Yaskawa INFORM job: X4-SCHODKI_ZEW.JBI

/JOB
//NAME X4-SCHODKI_ZEW
//POS
///NPOS 224,224,224,10,0,0
///TOOL 0
///POSTYPE PULSE
///PULSE
C00000=21160,-126487,-99095,6220,53097,19917
C00001=122314,-84956,-84267,5758,65294,20346
C00002=113867,-2788,-32259,11364,77586,-20622
C00003=111699,9606,-11794,12514,71800,-21939
C00004=110873,16102,-4909,12893,71047,-22311
C00005=111426,18220,-2948,12689,70847,-22135
C00006=111334,17863,-3281,12723,70881,-22164
C00007=111334,17842,-1921,12786,70054,-22254
C00008=111688,13758,-7042,12574,71029,-22022
C00009=137921,23655,2193,-26065,80546,13065
C00010=138187,30095,8478,-26164,80127,13260
C00011=137141,31636,10013,-25924,79665,12972
C00012=137283,31426,9804,-25956,79727,13011
C00013=137283,31447,11085,-26011,79025,13166
C00014=137811,24810,3269,-26040,80453,13045
C00015=130093,15204,-5597,-17076,73087,3422
C00016=130254,16762,-4164,-17139,73044,3486
C00017=130499,11823,-8660,-17205,73314,3535
C00018=136657,16032,-4835,-19303,74485,5576
C00019=136779,34044,12201,-19450,73350,5806
C00020=136367,37287,16065,-19383,72578,5782
C00021=135529,38270,17077,-19116,72272,5524
C00022=135735,38345,17156,-19186,72312,5593
C00023=135735,38391,18179,-19247,71738,5687
C00024=136093,38073,17157,-19317,72259,5733
C00025=136821,38987,18103,-19565,72324,5991
C00026=137234,41236,20445,-19732,72152,6174
C00027=137468,37941,16529,-19737,72884,6137
C00028=139273,33119,8814,-10616,74138,14432
C00029=138400,39162,15428,-10360,73077,14220
C00030=137624,40756,17090,-10099,72782,13973
C00031=137810,40443,16764,-10163,72844,14033
C00032=137810,40460,18419,-10216,71849,14119
C00033=138377,33107,10032,-10341,73283,14197
C00034=129933,32626,9546,1459,71562,3103
C00035=130107,34413,11352,1398,71367,3162
C00036=130344,28976,5916,1305,71915,3250
C00037=134876,30968,7890,-396,71698,4822
C00038=142592,70732,50995,-12851,68399,16892
C00039=141830,71409,51797,-12602,68137,16639
C00040=142006,70894,51186,-12652,68274,16689
C00041=142006,71149,52557,-12712,67578,16765
C00042=142006,71007,51815,-12679,67954,16725
C00043=142747,76515,58410,-13043,66871,17119
C00044=142702,66110,44987,-12780,69711,16790
C00045=130401,22900,-3912,9781,74013,14096
C00046=130750,-77898,-76934,10038,67211,13654
C00047=128341,-94500,-64478,15665,37561,8814
C00048=125354,-34494,-33676,16070,41961,8103
C00049=123908,-22688,-35224,-7311,60763,8117
C00050=115329,1774,-22996,-8583,68206,33205
C00051=113811,6923,-16554,-7934,66753,32769
C00052=112938,8598,-15088,-7517,66630,32466
C00053=113357,7607,-15958,-7718,66694,32611
C00054=113357,7474,-14642,-7767,65823,32669
C00055=113357,7562,-15559,-7732,66427,32629
C00056=114674,8046,-17033,-9196,71995,10105
C00057=114277,9137,-16073,-9034,71921,9973
C00058=114994,10710,-14679,-9331,71949,10219
C00059=115929,5782,-19714,-10610,72890,11247
C00060=114914,9168,-18033,-20160,83408,25507
C00061=114509,10465,-16323,-20060,82947,25443
C00062=114509,10278,-15209,-20089,82211,25564
C00063=114509,10430,-16126,-20066,82816,25464
C00064=113574,12027,-14696,-19812,82540,25184
C00065=113966,9476,-16971,-19916,82715,25292
C00066=109195,41890,2270,-19889,88323,22522
C00067=109420,41611,2136,-14547,83651,24420
C00068=109633,43097,3705,-14621,83493,24508
C00069=110073,47498,8361,-9922,80898,20177
C00070=110340,48514,8983,-10012,81065,20250
C00071=109875,50139,10594,-6927,80049,17487
C00072=111642,41129,-2073,-7513,83338,17864
C00073=120740,-4591,-30289,-15267,55452,23675
C00074=120758,-111403,-89341,-20679,37744,27189
C00075=120758,-111403,-89341,-20679,37744,27189
C00076=97140,-41370,-74515,11864,90116,-15742
C00077=93918,-16818,-51601,15265,90472,-19448
C00078=96838,-21310,-54909,14446,89719,-18600
C00079=97144,-22320,-55662,14359,89616,-18514
C00080=98771,-24881,-57497,13895,89173,-18041
C00081=115828,-29996,-61044,-7286,86100,2495
C00082=121364,-24267,-57094,-13933,89260,9154
C00083=125066,-13537,-49221,-14991,90516,10198
C00084=125405,-12324,-48437,-15087,90711,10281
C00085=127775,-3453,-41245,-15747,91251,10973
C00086=117906,-11103,-47413,-1372,86513,-3179
C00087=107817,-4833,-42392,13913,90158,-17947
C00088=111065,-8601,-45456,12965,89620,-16971
C00089=111228,-9142,-45834,12917,89553,-16926
C00090=113235,-11504,-47787,12324,89257,-16321
C00091=116129,-16038,-53218,11461,89860,-15351
C00092=132129,3503,-37461,731,88042,-5165
C00093=134839,10104,-29765,-1476,86561,-3078
C00094=133535,10494,-29542,-1044,86604,-3481
C00095=133472,10527,-29512,-1023,86602,-3500
C00096=132997,13157,-27039,-5636,86965,851
C00097=131112,-12606,-50888,-7793,88905,29033
C00098=129834,-10958,-47906,-7386,87816,28703
C00099=133351,1378,-37957,-8503,88347,29764
C00100=133639,2898,-36665,-8594,88358,29852
C00101=132895,14544,-26435,-2898,86896,24452
C00102=133144,15405,-25686,-2979,86883,24528
C00103=133588,9909,-35564,-3125,90148,24585
C00104=114600,-38617,-66572,24501,76796,21744
C00105=88804,-102668,-113384,34072,81784,13502
C00106=-3643,-76224,-106676,-19950,71810,-76872
C00107=-6047,-95755,-92046,14751,98253,-9605
C00108=-2299,-70459,-84112,3705,91093,-18065
C00109=-2299,-70459,-84112,3705,91093,-18065
C00110=-2299,-70459,-84112,3705,91093,-18065
C00111=-2299,-70459,-84112,3705,91093,-18065
C00112=61951,-108908,-90353,7974,21769,-53190
C00113=44975,-75191,-76287,54105,62461,-71292
C00114=78581,-58710,-61930,31634,35162,-55381
C00115=95060,-56001,-58325,12610,29924,-73279
C00116=99699,-51031,-54888,6140,29822,-70179
C00117=99897,-48307,-53304,5791,30229,-70010
C00118=100054,-49149,-53798,5600,30089,-69920
C00119=100054,-49034,-52503,5728,29355,-69986
C00120=100054,-49149,-53798,5600,30089,-69920
C00121=86412,-51164,-57714,27133,38899,-75152
C00122=76272,-10487,-35891,41089,67840,-66679
C00123=77011,-10638,-36009,40769,67508,-66483
C00124=76817,-10362,-35793,40851,67601,-66531
C00125=76817,-10560,-34912,41019,67109,-66737
C00126=76817,-10362,-35793,40851,67601,-66531
C00127=75718,7442,-20978,41322,68120,-66813
C00128=76464,7847,-20622,41001,67775,-66619
C00129=76126,7559,-20874,41146,67933,-66706
C00130=76126,7348,-19931,41325,67409,-66927
C00131=76126,7559,-20874,41146,67933,-66706
C00132=91627,-14375,-38555,867,50575,-46141
C00133=91624,-12364,-37017,870,50664,-46141
C00134=91625,-13152,-37622,869,50631,-46141
C00135=91625,-13360,-36631,878,49914,-46147
C00136=91625,-13152,-37622,869,50631,-46141
C00137=68864,9101,-19550,42290,68970,-68812
C00138=70480,17607,-11844,41698,67948,-68513
C00139=71103,18297,-11202,41441,67635,-68362
C00140=70696,17763,-11700,41608,67844,-68460
C00141=70696,17560,-10741,41791,67318,-68687
C00142=70696,17763,-11700,41608,67844,-68460
C00143=71865,37445,7605,38393,62836,-66759
C00144=72519,37882,8057,38094,62514,-66586
C00145=71865,37445,7605,38393,62836,-66759
C00146=71865,37288,8698,38629,62241,-66997
C00147=71865,37445,7605,38393,62836,-66759
C00148=69589,28187,-3550,38858,65482,-66746
C00149=81736,18570,-13478,9629,55098,-51480
C00150=92480,21393,-8443,-18166,53536,-36270
C00151=92406,23699,-6245,-18150,53360,-36270
C00152=92480,21393,-8443,-18166,53536,-36270
C00153=92480,21153,-7249,-18365,52720,-36120
C00154=92480,21393,-8443,-18166,53536,-36270
C00155=66161,2763,-24906,35901,59847,-65565
C00156=8779,-64345,-72223,57070,85976,-80913
C00157=8779,-64345,-72223,57070,85976,-80913
C00158=80709,2938,-29836,37807,72072,-57205
C00159=104099,16313,-17981,36138,70132,-56262
C00160=141757,27909,-6366,14089,61839,-44283
C00161=141757,27617,-5405,14183,61121,-44376
C00162=141757,27909,-6366,14089,61839,-44283
C00163=142084,29535,-4762,13913,61639,-44186
C00164=141757,27909,-6366,14089,61839,-44283
C00165=134298,42766,7339,18583,62496,-46981
C00166=136587,44887,8503,12300,63619,-46934
C00167=136587,44658,9247,12359,63057,-46997
C00168=136587,44887,8503,12300,63619,-46934
C00169=137255,47131,10909,11951,63202,-46735
C00170=136587,44887,8503,12300,63619,-46934
C00171=137657,47095,11743,9838,62197,-45465
C00172=138989,44169,8634,9022,62453,-44958
C00173=139465,42914,7769,8751,62290,-44797
C00174=139736,38942,3601,15550,64524,-48931
C00175=140033,37764,2383,15370,64612,-48812
C00176=142152,32374,-3332,17000,65924,-49772
C00177=136320,25956,-14717,19617,70677,-51083
C00178=115846,-52963,-75028,29682,73275,-57924
C00179=37442,-83575,-86281,52659,88245,-87706
C00180=33903,-112886,-95665,42735,53090,-80159
C00181=69561,-59751,-72923,16095,52051,-63361
C00182=88044,4124,-27726,-14416,55568,-38396
C00183=89480,30550,-2469,-15773,59241,-38542
C00184=89566,29946,-3118,-13987,58895,-39575
C00185=89868,30274,-2806,-13508,58764,-39848
C00186=89813,28581,-4483,-7975,57782,-42956
C00187=83888,29903,-3137,7775,57604,-51754
C00188=72316,13965,-19527,34407,71386,-67147
C00189=73909,13977,-18764,33784,70394,-66825
C00190=73971,16364,-16409,33799,70187,-66867
C00191=73672,28324,-4910,34113,69520,-67204
C00192=73857,29288,-3960,34049,69373,-67175
C00193=73190,47231,14588,34804,67803,-67970
C00194=76539,39499,6435,26306,62774,-62506
C00195=71407,-68,-33227,28174,68008,-63188
C00196=92287,-5015,-35072,-6189,59116,-43997
C00197=93582,-5318,-35114,-7054,59088,-43517
C00198=94768,-5424,-35240,-7833,59212,-43086
C00199=95122,-4999,-34965,-8061,59297,-42962
C00200=98977,-4910,-34893,-10570,59720,-41566
C00201=89817,-2997,-33375,10480,59755,-53225
C00202=87165,-16267,-43774,12233,59696,-54222
C00203=74457,-13339,-39679,39309,71456,-68037
C00204=78370,-12635,-39382,37625,69939,-66937
C00205=80519,-10300,-39984,32672,71010,-66549
C00206=79797,2903,-29087,32982,71339,-66737
C00207=79943,3599,-28462,32921,71264,-66703
C00208=82505,7061,-25304,26471,66621,-62758
C00209=86409,1492,-30136,17739,62740,-57641
C00210=82783,-10794,-40788,19813,63755,-58809
C00211=89567,-44228,-57976,15859,46252,-64914
C00212=95371,-48907,-52544,12165,29960,-73065
C00213=96871,-48956,-52574,10129,29748,-72091
C00214=98013,-48924,-52556,8555,29621,-71337
C00215=98537,-48530,-52441,7796,29699,-70974
C00216=102207,-48035,-52053,2674,29480,-68529
C00217=94327,-44885,-50172,28699,34004,-81028
C00218=94609,-45389,-50476,28446,33845,-80908
C00219=90036,-53113,-58492,32420,36321,-82805
C00220=51114,-81290,-74278,61960,52593,-60278
C00221=6076,-109546,-85200,71251,79672,-70600
C00222=6076,-109546,-85200,71251,79672,-70600
C00223=6076,-109546,-85200,-4239,76823,-70600
BC00000=277643,516186,172088
BC00001=328181,496789,172088
BC00002=328180,496788,172085
BC00003=328180,496788,172085
BC00004=328180,496788,172085
BC00005=328180,496788,172085
BC00006=328180,496788,172085
BC00007=328180,496788,172085
BC00008=328180,496788,172085
BC00009=328180,496788,172085
BC00010=328180,496788,172085
BC00011=328180,496788,172085
BC00012=328180,496788,172085
BC00013=328180,496788,172085
BC00014=328180,496788,172085
BC00015=328180,496788,172085
BC00016=328180,496788,172085
BC00017=328180,496788,172085
BC00018=328180,496788,172085
BC00019=328180,496788,172085
BC00020=328180,496788,172085
BC00021=328180,496788,172085
BC00022=328180,496788,172085
BC00023=328180,496788,172085
BC00024=328180,496788,172085
BC00025=328180,496788,172085
BC00026=328180,496788,172085
BC00027=328180,496788,172085
BC00028=328180,496788,172085
BC00029=328180,496788,172085
BC00030=328180,496788,172085
BC00031=328180,496788,172085
BC00032=328180,496788,172085
BC00033=328180,496788,172085
BC00034=328180,496788,172085
BC00035=328180,496788,172085
BC00036=328180,496788,172085
BC00037=328180,496788,172085
BC00038=328180,496788,172085
BC00039=328180,496788,172085
BC00040=328180,496788,172085
BC00041=328180,496788,172085
BC00042=328180,496788,172085
BC00043=328180,496788,172085
BC00044=328180,496788,172085
BC00045=328180,496788,172085
BC00046=328180,496788,172085
BC00047=194416,502028,172085
BC00048=194416,502028,172085
BC00049=173311,425006,172085
BC00050=173311,425006,140819
BC00051=173311,425006,140819
BC00052=173311,425006,140819
BC00053=173311,425006,140819
BC00054=173311,425006,140819
BC00055=173311,425006,140819
BC00056=173311,425006,140819
BC00057=173311,425006,140819
BC00058=173311,425006,140819
BC00059=173311,425006,140819
BC00060=173311,425006,140819
BC00061=173311,425006,140819
BC00062=173311,425006,140819
BC00063=173311,425006,140819
BC00064=173311,425006,140819
BC00065=173311,425006,140819
BC00066=158492,452266,59327
BC00067=158492,452266,59327
BC00068=158492,452266,59327
BC00069=158492,452266,59327
BC00070=158492,452266,59327
BC00071=158492,452266,59327
BC00072=158492,452266,59327
BC00073=158492,452266,59327
BC00074=158492,507957,59327
BC00075=293306,507957,59327
BC00076=293305,437676,59324
BC00077=293305,437676,59324
BC00078=293305,437676,59324
BC00079=293305,437676,59324
BC00080=293305,437676,59324
BC00081=293305,437676,59324
BC00082=293305,437676,59324
BC00083=293305,437676,59324
BC00084=293305,437676,59324
BC00085=293305,437676,59324
BC00086=293305,437676,59324
BC00087=293305,437676,59324
BC00088=293305,437676,59324
BC00089=293305,437676,59324
BC00090=293305,437676,59324
BC00091=293305,437676,59324
BC00092=293305,437676,59324
BC00093=293305,437676,59324
BC00094=293305,437676,59324
BC00095=293305,437676,59324
BC00096=293305,437676,59324
BC00097=293305,437676,59324
BC00098=293305,437676,59324
BC00099=293305,437676,59324
BC00100=293305,437676,59324
BC00101=293305,437676,59324
BC00102=293305,437676,59324
BC00103=293305,437676,59324
BC00104=293305,437676,59324
BC00105=293305,491548,59324
BC00106=199448,515539,1075137
BC00107=95028,515070,919110
BC00108=123826,515279,972180
BC00109=123826,515279,972180
BC00110=123826,515279,972180
BC00111=44761,462630,27794
BC00112=44761,462630,27794
BC00113=44761,462630,27793
BC00114=44761,462630,27793
BC00115=44761,462630,27793
BC00116=44761,462630,27793
BC00117=44761,462630,27793
BC00118=44761,462630,27793
BC00119=44761,462630,27793
BC00120=44761,462630,27793
BC00121=44761,462630,27793
BC00122=44761,462630,27793
BC00123=44761,462630,27793
BC00124=44761,462630,27793
BC00125=44761,462630,27793
BC00126=44761,462630,27793
BC00127=44761,462630,27793
BC00128=44761,462630,27793
BC00129=44761,462630,27793
BC00130=44761,462630,27793
BC00131=44761,462630,27793
BC00132=44761,462630,27793
BC00133=44761,462630,27793
BC00134=44761,462630,27793
BC00135=44761,462630,27793
BC00136=44761,462630,27793
BC00137=44761,462630,27793
BC00138=44761,462630,27793
BC00139=44761,462630,27793
BC00140=44761,462630,27793
BC00141=44761,462630,27793
BC00142=44761,462630,27793
BC00143=44761,462630,27793
BC00144=44761,462630,27793
BC00145=44761,462630,27793
BC00146=44761,462630,27793
BC00147=44761,462630,27793
BC00148=44761,462630,27793
BC00149=44761,462630,27793
BC00150=44761,462630,27793
BC00151=44761,462630,27793
BC00152=44761,462630,27793
BC00153=44761,462630,27793
BC00154=44761,462630,27793
BC00155=44761,462630,27792
BC00156=44761,462630,27792
BC00157=202931,462630,27792
BC00158=202931,462630,27792
BC00159=222940,462630,27792
BC00160=308656,462630,27792
BC00161=308656,462630,27792
BC00162=308656,462630,27792
BC00163=308656,462630,27792
BC00164=308656,462630,27792
BC00165=308656,462630,27792
BC00166=308656,462630,27792
BC00167=308656,462630,27792
BC00168=308656,462630,27792
BC00169=308656,462630,27792
BC00170=308656,462630,27792
BC00171=308656,462630,27792
BC00172=308656,462630,27792
BC00173=308656,462630,27792
BC00174=308656,462630,27792
BC00175=308656,462630,27792
BC00176=308656,462630,27792
BC00177=308656,462630,27792
BC00178=308656,462630,27791
BC00179=194109,459376,27791
BC00180=59950,457329,27792
BC00181=59950,457329,27792
BC00182=44761,462630,27793
BC00183=44761,462629,27792
BC00184=44761,462629,27792
BC00185=44761,462629,27792
BC00186=44761,462629,27792
BC00187=44761,462629,27792
BC00188=44761,462629,27792
BC00189=44761,462629,27792
BC00190=44761,462629,27792
BC00191=44761,462629,27792
BC00192=44761,462629,27792
BC00193=44761,462629,27792
BC00194=44761,462629,27792
BC00195=44761,462629,27792
BC00196=44761,462629,27792
BC00197=44761,462629,27792
BC00198=44761,462629,27792
BC00199=44761,462629,27792
BC00200=44761,462629,27792
BC00201=44761,462629,27792
BC00202=44761,462629,27792
BC00203=44761,462629,27792
BC00204=44761,462629,27792
BC00205=44761,462629,27792
BC00206=44761,462629,27792
BC00207=44761,462629,27792
BC00208=44761,462629,27792
BC00209=44761,462629,27792
BC00210=44761,462629,27792
BC00211=44761,462629,27792
BC00212=44761,462630,27793
BC00213=44761,462630,27793
BC00214=44761,462630,27793
BC00215=44761,462630,27793
BC00216=44761,462630,27793
BC00217=44761,462630,27793
BC00218=44761,462630,27793
BC00219=44761,462630,27793
BC00220=44761,462630,27793
BC00221=44761,546100,27793
BC00222=44761,546100,27793
BC00223=44761,546100,971290
EC00000=798156,-183832
EC00001=798156,-183832
EC00002=798153,-183831
EC00003=798153,-183831
EC00004=798153,-183831
EC00005=798153,-183831
EC00006=798153,-183831
EC00007=798153,-183831
EC00008=798153,-183831
EC00009=798153,-183831
EC00010=798153,-183831
EC00011=798153,-183831
EC00012=798153,-183831
EC00013=798153,-183831
EC00014=798153,-183831
EC00015=798153,-183831
EC00016=798153,-183831
EC00017=798153,-183831
EC00018=798153,-183831
EC00019=798153,-183831
EC00020=798153,-183831
EC00021=798153,-183831
EC00022=798153,-183831
EC00023=798153,-183831
EC00024=798153,-183831
EC00025=798153,-183831
EC00026=798153,-183831
EC00027=798153,-183831
EC00028=798153,-183831
EC00029=798153,-183831
EC00030=798153,-183831
EC00031=798153,-183831
EC00032=798153,-183831
EC00033=798153,-183831
EC00034=798153,-183831
EC00035=798153,-183831
EC00036=798153,-183831
EC00037=798153,-183831
EC00038=798153,-183831
EC00039=798153,-183831
EC00040=798153,-183831
EC00041=798153,-183831
EC00042=798153,-183831
EC00043=798153,-183831
EC00044=798153,-183831
EC00045=798153,-183831
EC00046=798153,-183831
EC00047=798153,-183831
EC00048=798153,-183831
EC00049=798153,-183831
EC00050=798153,-183831
EC00051=798153,-183831
EC00052=798153,-183831
EC00053=798153,-183831
EC00054=798153,-183831
EC00055=798153,-183831
EC00056=798153,-183831
EC00057=798153,-183831
EC00058=798153,-183831
EC00059=798153,-183831
EC00060=798153,-183831
EC00061=798153,-183831
EC00062=798153,-183831
EC00063=798153,-183831
EC00064=798153,-183831
EC00065=798153,-183831
EC00066=798153,-183831
EC00067=798153,-183831
EC00068=798153,-183831
EC00069=798153,-183831
EC00070=798153,-183831
EC00071=798153,-183831
EC00072=798153,-183831
EC00073=798153,-183831
EC00074=798153,-183831
EC00075=798153,-183831
EC00076=798151,-183830
EC00077=798151,-183830
EC00078=798151,-183830
EC00079=798151,-183830
EC00080=798151,-183830
EC00081=798151,-183830
EC00082=798151,-183830
EC00083=798151,-183830
EC00084=798151,-183830
EC00085=798151,-183830
EC00086=798151,-183830
EC00087=798151,-183830
EC00088=798151,-183830
EC00089=798151,-183830
EC00090=798151,-183830
EC00091=798151,-183830
EC00092=798151,-183830
EC00093=798151,-183830
EC00094=798151,-183830
EC00095=798151,-183830
EC00096=798151,-183830
EC00097=798151,-183830
EC00098=798151,-183830
EC00099=798151,-183830
EC00100=798151,-183830
EC00101=798151,-183830
EC00102=798151,-183830
EC00103=798151,-183830
EC00104=798151,-183830
EC00105=798151,-183830
EC00106=798151,-183830
EC00107=798156,-183832
EC00108=322978,-183832
EC00109=357094,925242
EC00110=800604,925242
EC00111=800604,925242
EC00112=800604,925242
EC00113=800603,925242
EC00114=800603,925242
EC00115=800603,925242
EC00116=800603,925242
EC00117=800603,925242
EC00118=800603,925242
EC00119=800603,925242
EC00120=800603,925242
EC00121=800603,925242
EC00122=800603,925242
EC00123=800603,925242
EC00124=800603,925242
EC00125=800603,925242
EC00126=800603,925242
EC00127=800603,925242
EC00128=800603,925242
EC00129=800603,925242
EC00130=800603,925242
EC00131=800603,925242
EC00132=800603,925242
EC00133=800603,925242
EC00134=800603,925242
EC00135=800603,925242
EC00136=800603,925242
EC00137=800603,925242
EC00138=800603,925242
EC00139=800603,925242
EC00140=800603,925242
EC00141=800603,925242
EC00142=800603,925242
EC00143=800603,925242
EC00144=800603,925242
EC00145=800603,925242
EC00146=800603,925242
EC00147=800603,925242
EC00148=800603,925242
EC00149=800601,925240
EC00150=800600,925239
EC00151=800600,925239
EC00152=800600,925239
EC00153=800600,925239
EC00154=800600,925239
EC00155=800598,925238
EC00156=800598,925238
EC00157=800598,925238
EC00158=800598,925238
EC00159=800598,925238
EC00160=800598,925238
EC00161=800598,925238
EC00162=800598,925238
EC00163=800598,925238
EC00164=800598,925238
EC00165=800598,925238
EC00166=800598,925238
EC00167=800598,925238
EC00168=800598,925238
EC00169=800598,925238
EC00170=800598,925238
EC00171=800598,925238
EC00172=800598,925238
EC00173=800598,925238
EC00174=800598,925238
EC00175=800598,925238
EC00176=800598,925238
EC00177=800598,925238
EC00178=800591,925233
EC00179=800591,925233
EC00180=800596,925236
EC00181=800596,925236
EC00182=800600,925239
EC00183=800597,925236
EC00184=800597,925236
EC00185=800597,925236
EC00186=800597,925236
EC00187=800597,925236
EC00188=800597,925236
EC00189=800597,925236
EC00190=800597,925236
EC00191=800597,925236
EC00192=800597,925236
EC00193=800597,925236
EC00194=800597,925236
EC00195=800597,925236
EC00196=800597,925236
EC00197=800597,925236
EC00198=800597,925236
EC00199=800597,925236
EC00200=800597,925236
EC00201=800597,925236
EC00202=800597,925236
EC00203=800597,925236
EC00204=800597,925236
EC00205=800597,925236
EC00206=800597,925236
EC00207=800597,925236
EC00208=800597,925236
EC00209=800597,925236
EC00210=800594,925234
EC00211=800598,925238
EC00212=800603,925242
EC00213=800603,925242
EC00214=800603,925242
EC00215=800603,925242
EC00216=800603,925242
EC00217=800603,925242
EC00218=800603,925242
EC00219=800603,925242
EC00220=800603,925242
EC00221=800603,925242
EC00222=-11362,925242
EC00223=-11362,925242
///POSTYPE BASE
///RECTAN
///RCONF 0,0,0,0,1,0,0,0,0,0,0,0,0,0,0,0,0,0,0,0,0,0,0,0
P00006=2.006,1.622,-0.565,0.0000,0.0000,0.0000
P00021=0.073,2.058,-0.109,0.0000,0.0000,0.0000
P00022=2.006,1.622,-0.565,0.0000,0.0000,0.0000
///RCONF 0,0,0,0,0,0,0,0,0,0,0,0,0,0,0,0,0,0,0,0,0,0,0,0
P00023=-2.957,-4.083,2.762,0.0000,0.0000,0.0000
P00024=-1.466,-0.226,-0.419,0.0000,0.0000,0.0000
P00025=3.643,0.007,-2.585,0.0000,0.0000,0.0000
P00026=2.644,0.055,-2.583,0.0000,0.0000,0.0000
P00027=2.278,0.099,-4.210,0.0000,0.0000,0.0000
P00028=-1.778,-0.182,-2.050,0.0000,0.0000,0.0000
P00029=1.749,4.006,-0.261,0.0000,0.0000,0.0000
//INST
///DATE 2024/11/26 12:08
///ATTR SC,RW
///GROUP1 RB1,BS1
///GROUP2 ST1
NOP
MOVJ C00000 BC00000 VJ=100.00  +MOVJ EC00000 VJ=100.00
MOVJ C00001 BC00001 VJ=100.00  +MOVJ EC00001 VJ=100.00
MOVJ C00002 BC00002 VJ=100.00  +MOVJ EC00002 VJ=100.00
SMOVL C00003 BC00003 V=833.3  +MOVJ EC00003
SMOVL C00004 BC00004 V=166.7  +MOVJ EC00004
SREFP 3 C00005 BC00005  +REFP EC00005
CALL JOB:SEARCH-R1-S13D
SET P021 P006
SFTON3D P021
SMOVL C00006 BC00006 V=166.7  +MOVJ EC00006
SREFP 3 C00007 BC00007  +REFP EC00007
CALL JOB:SEARCH-R1-S13D
SET P021 P006
SFTON3D P021
SMOVL C00008 BC00008 V=166.7  +MOVJ EC00008
SFTOF3D
SMOVL C00009 BC00009 V=833.3  +MOVJ EC00009
SMOVL C00010 BC00010 V=166.7  +MOVJ EC00010
SREFP 3 C00011 BC00011  +REFP EC00011
CALL JOB:SEARCH-R1-S13D
SET P022 P006
SFTON3D P022
SMOVL C00012 BC00012 V=166.7  +MOVJ EC00012
SREFP 3 C00013 BC00013  +REFP EC00013
CALL JOB:SEARCH-R1-S13D
SET P022 P006
SFTON3D P022
SMOVL C00014 BC00014 V=166.7  +MOVJ EC00014
SMOVL C00015 BC00015 V=166.7  +MOVJ EC00015
SREFP 3 C00016 BC00016  +REFP EC00016
CALL JOB:SEARCH-R1-S13D
SET P022 P006
SFTON3D P022
SMOVL C00017 BC00017 V=166.7  +MOVJ EC00017
SFTOF3D
SMOVL C00018 BC00018 V=500.0  +MOVJ EC00018
SMOVL C00019 BC00019 V=500.0  +MOVJ EC00019
SMOVL C00020 BC00020 V=166.7  +MOVJ EC00020
SREFP 3 C00021 BC00021  +REFP EC00021
CALL JOB:SEARCH-R1-S13D
SET P023 P006
SFTON3D P023
SMOVL C00022 BC00022 V=166.7  +MOVJ EC00022
SREFP 3 C00023 BC00023  +REFP EC00023
CALL JOB:SEARCH-R1-S13D
SET P023 P006
SFTON3D P023
SMOVL C00024 BC00024 V=166.7  +MOVJ EC00024
SMOVL C00025 BC00025 V=166.7  +MOVJ EC00025
SREFP 3 C00026 BC00026  +REFP EC00026
CALL JOB:SEARCH-R1-S13D
SET P023 P006
SFTON3D P023
SMOVL C00027 BC00027 V=166.7  +MOVJ EC00027
SFTOF3D
SMOVL C00028 BC00028 V=333.3  +MOVJ EC00028
SMOVL C00029 BC00029 V=166.7  +MOVJ EC00029
SREFP 3 C00030 BC00030  +REFP EC00030
CALL JOB:SEARCH-R1-S13D
SET P024 P006
SFTON3D P024
SMOVL C00031 BC00031 V=166.7  +MOVJ EC00031
SREFP 3 C00032 BC00032  +REFP EC00032
CALL JOB:SEARCH-R1-S13D
SET P024 P006
SFTON3D P024
SMOVL C00033 BC00033 V=166.7  +MOVJ EC00033
SMOVL C00034 BC00034 V=166.7  +MOVJ EC00034
SREFP 3 C00035 BC00035  +REFP EC00035
CALL JOB:SEARCH-R1-S13D
SET P024 P006
SFTON3D P024
SMOVL C00036 BC00036 V=166.7  +MOVJ EC00036
SFTOF3D
SMOVL C00037 BC00037 V=333.3  +MOVJ EC00037
SMOVL C00038 BC00038 V=166.7  +MOVJ EC00038
SREFP 3 C00039 BC00039  +REFP EC00039
CALL JOB:SEARCH-R1-S13D
SET P025 P006
SFTON3D P025
SMOVL C00040 BC00040 V=166.7  +MOVJ EC00040
SREFP 3 C00041 BC00041  +REFP EC00041
CALL JOB:SEARCH-R1-S13D
SET P025 P006
SFTON3D P025
SMOVL C00042 BC00042 V=166.7  +MOVJ EC00042
SREFP 3 C00043 BC00043  +REFP EC00043
CALL JOB:SEARCH-R1-S13D
SET P025 P006
SFTON3D P025
SMOVL C00044 BC00044 V=166.7  +MOVJ EC00044
SFTOF3D
SMOVL C00045 BC00045 V=333.3  +MOVJ EC00045
SMOVL C00046 BC00046 V=1000.0  +MOVJ EC00046
SMOVL C00047 BC00047 V=1000.0  +MOVJ EC00047
SMOVL C00048 BC00048 V=1000.0  +MOVJ EC00048
SMOVL C00049 BC00049 V=666.7  +MOVJ EC00049
SMOVL C00050 BC00050 V=666.7  +MOVJ EC00050
SMOVL C00051 BC00051 V=166.7  +MOVJ EC00051
SREFP 3 C00052 BC00052  +REFP EC00052
CALL JOB:SEARCH-R1-S13D
SET P027 P006
SFTON3D P027
SMOVL C00053 BC00053 V=166.7  +MOVJ EC00053
SREFP 3 C00054 BC00054  +REFP EC00054
CALL JOB:SEARCH-R1-S13D
SET P027 P006
SFTON3D P027
SMOVL C00055 BC00055 V=166.7  +MOVJ EC00055
SMOVL C00056 BC00056 V=250.0  +MOVJ EC00056
SMOVL C00057 BC00057 V=250.0  +MOVJ EC00057
SREFP 3 C00058 BC00058  +REFP EC00058
CALL JOB:SEARCH-R1-S13D
SET P027 P006
SFTON3D P027
SMOVL C00059 BC00059 V=166.7  +MOVJ EC00059
SFTOF3D
SMOVL C00060 BC00060 V=250.0  +MOVJ EC00060
SMOVL C00061 BC00061 V=166.7  +MOVJ EC00061
SREFP 3 C00062 BC00062  +REFP EC00062
CALL JOB:SEARCH-R1-S13D
SET P026 P006
SFTON3D P026
SMOVL C00063 BC00063 V=166.7  +MOVJ EC00063
SREFP 3 C00064 BC00064  +REFP EC00064
CALL JOB:SEARCH-R1-S13D
SET P026 P006
SFTON3D P026
SMOVL C00065 BC00065 V=166.7  +MOVJ EC00065
MACRO1 MJ#(0) ARGF9
SMOVL C00066 BC00066 V=250.0  +MOVJ EC00066
ARCON
SMOVL C00067 BC00067 V=10.0  +MOVJ EC00067
SMOVL C00068 BC00068 V=10.0  +MOVJ EC00068
SFTON3D P027
SMOVL C00069 BC00069 V=10.0  +MOVJ EC00069
ARCOF
SMOVL C00070 BC00070 V=10.0  +MOVJ EC00070
ARCON
SMOVL C00071 BC00071 V=10.0  +MOVJ EC00071
ARCOF
SFTOF3D
SMOVL C00072 BC00072 V=250.0  +MOVJ EC00072
SMOVL C00073 BC00073 V=666.7  +MOVJ EC00073
SMOVL C00074 BC00074 V=666.7  +MOVJ EC00074
SMOVL C00075 BC00075 V=1000.0  +MOVJ EC00075
SMOVL C00076 BC00076 V=1000.0  +MOVJ EC00076
SFTON3D P021
SMOVL C00077 BC00077 V=166.7  +MOVJ EC00077
ARCON
SMOVL C00078 BC00078 V=10.0  +MOVJ EC00078
SFTON3D P022
SMOVL C00079 BC00079 V=10.0  +MOVJ EC00079
SMOVL C00080 BC00080 V=10.0  +MOVJ EC00080
SMOVL C00081 BC00081 V=10.0  +MOVJ EC00081
SMOVL C00082 BC00082 V=10.0  +MOVJ EC00082
SMOVL C00083 BC00083 V=10.0  +MOVJ EC00083
SMOVL C00084 BC00084 V=10.0  +MOVJ EC00084
SFTON3D P023
SMOVL C00085 BC00085 V=10.0  +MOVJ EC00085
SMOVL C00086 BC00086 V=10.0  +MOVJ EC00086
SMOVL C00087 BC00087 V=10.0  +MOVJ EC00087
SMOVL C00088 BC00088 V=10.0  +MOVJ EC00088
SFTON3D P024
SMOVL C00089 BC00089 V=10.0  +MOVJ EC00089
SMOVL C00090 BC00090 V=10.0  +MOVJ EC00090
ARCOF
SFTOF3D
SMOVL C00091 BC00091 V=250.0  +MOVJ EC00091
SMOVL C00092 BC00092 V=500.0  +MOVJ EC00092
SFTON3D P026
SMOVL C00093 BC00093 V=250.0  +MOVJ EC00093
ARCON
SMOVL C00094 BC00094 V=10.0  +MOVJ EC00094
SMOVL C00095 BC00095 V=10.0  +MOVJ EC00095
SFTON3D P025
SMOVL C00096 BC00096 V=10.0  +MOVJ EC00096
ARCOF
SFTOF3D
SMOVL C00097 BC00097 V=400.0  +MOVJ EC00097
SFTON3D P024
SMOVL C00098 BC00098 V=166.7  +MOVJ EC00098
ARCON
SMOVL C00099 BC00099 V=10.0  +MOVJ EC00099
SMOVL C00100 BC00100 V=10.0  +MOVJ EC00100
SFTON3D P025
SMOVL C00101 BC00101 V=10.0  +MOVJ EC00101
SMOVL C00102 BC00102 V=10.0  +MOVJ EC00102
ARCOF
SFTOF3D
SMOVL C00103 BC00103 V=250.0  +MOVJ EC00103
SMOVL C00104 BC00104 V=833.3  +MOVJ EC00104
MOVJ C00105 BC00105 VJ=100.00  +MOVJ EC00105 VJ=100.00
MOVJ C00106 BC00106 VJ=100.00  +MOVJ EC00106 VJ=100.00
CALL JOB:CLEAN-R1_KM_NEW
MOVJ C00107 BC00107 VJ=100.00  +MOVJ EC00107 VJ=100.00
PAUSE
MOVJ C00108 BC00108 VJ=100.00  +MOVJ EC00108 VJ=100.00
MOVJ C00109 BC00109 VJ=100.00  +MOVJ EC00109 VJ=100.00
MOVJ C00110 BC00110 VJ=100.00  +MOVJ EC00110 VJ=100.00
MOVJ C00111 BC00111 VJ=100.00  +MOVJ EC00111 VJ=100.00
MOVJ C00112 BC00112 VJ=100.00  +MOVJ EC00112 VJ=100.00
MOVJ C00113 BC00113 VJ=30.00  +MOVJ EC00113 VJ=100.00
MOVL C00114 BC00114 V=333.3  +MOVJ EC00114 VJ=30.00
MOVL C00115 BC00115 V=333.3  +MOVJ EC00115 VJ=30.00
SFTOF3D
SMOVL C00116 BC00116 V=166.7  +MOVJ EC00116
SREFP 3 C00117 BC00117  +REFP EC00117
CALL JOB:SEARCH-R1-S13D
SET P027 P006
SFTON3D P027
SMOVL C00118 BC00118 V=166.7  +MOVJ EC00118
SREFP 3 C00119 BC00119  +REFP EC00119
CALL JOB:SEARCH-R1-S13D
SET P027 P006
SFTON3D P027
SMOVL C00120 BC00120 V=166.7  +MOVJ EC00120
SFTOF3D
MOVL C00121 BC00121 V=333.3  +MOVJ EC00121 VJ=30.00
SFTOF3D
SMOVL C00122 BC00122 V=166.7  +MOVJ EC00122
SREFP 3 C00123 BC00123  +REFP EC00123
CALL JOB:SEARCH-R1-S13D
SET P026 P006
SFTON3D P026
SMOVL C00124 BC00124 V=166.7  +MOVJ EC00124
SREFP 3 C00125 BC00125  +REFP EC00125
CALL JOB:SEARCH-R1-S13D
SET P026 P006
SFTON3D P026
SMOVL C00126 BC00126 V=166.7  +MOVJ EC00126
SFTOF3D
SMOVL C00127 BC00127 V=166.7  +MOVJ EC00127
SREFP 3 C00128 BC00128  +REFP EC00128
CALL JOB:SEARCH-R1-S13D
SET P025 P006
SFTON3D P025
SMOVL C00129 BC00129 V=166.7  +MOVJ EC00129
SREFP 3 C00130 BC00130  +REFP EC00130
CALL JOB:SEARCH-R1-S13D
SET P025 P006
SFTON3D P025
SMOVL C00131 BC00131 V=166.7  +MOVJ EC00131
SFTOF3D
SMOVL C00132 BC00132 V=166.7  +MOVJ EC00132
SREFP 3 C00133 BC00133  +REFP EC00133
CALL JOB:SEARCH-R1-S13D
SET P024 P006
SFTON3D P024
SMOVL C00134 BC00134 V=166.7  +MOVJ EC00134
SREFP 3 C00135 BC00135  +REFP EC00135
CALL JOB:SEARCH-R1-S13D
SET P024 P006
SFTON3D P024
SMOVL C00136 BC00136 V=166.7  +MOVJ EC00136
SFTOF3D
MOVL C00137 BC00137 V=333.3  +MOVJ EC00137 VJ=30.00
SMOVL C00138 BC00138 V=166.7  +MOVJ EC00138
SREFP 3 C00139 BC00139  +REFP EC00139
CALL JOB:SEARCH-R1-S13D
SET P028 P006
SFTON3D P028
SMOVL C00140 BC00140 V=166.7  +MOVJ EC00140
SREFP 3 C00141 BC00141  +REFP EC00141
CALL JOB:SEARCH-R1-S13D
SET P028 P006
SFTON3D P028
SMOVL C00142 BC00142 V=166.7  +MOVJ EC00142
SFTOF3D
SMOVL C00143 BC00143 V=166.7  +MOVJ EC00143
SREFP 3 C00144 BC00144  +REFP EC00144
CALL JOB:SEARCH-R1-S13D
SET P023 P006
SFTON3D P023
SMOVL C00145 BC00145 V=166.7  +MOVJ EC00145
SREFP 3 C00146 BC00146  +REFP EC00146
CALL JOB:SEARCH-R1-S13D
SET P023 P006
SFTON3D P023
SMOVL C00147 BC00147 V=166.7  +MOVJ EC00147
SFTOF3D
MOVJ C00148 BC00148 VJ=30.00  +MOVJ EC00148 VJ=30.00
MOVJ C00149 BC00149 VJ=30.00  +MOVJ EC00149 VJ=30.00
SMOVL C00150 BC00150 V=166.7  +MOVJ EC00150
SREFP 3 C00151 BC00151  +REFP EC00151
CALL JOB:SEARCH-R1-S13D
SET P029 P006
SFTON3D P029
SMOVL C00152 BC00152 V=166.7  +MOVJ EC00152
SREFP 3 C00153 BC00153  +REFP EC00153
CALL JOB:SEARCH-R1-S13D
SET P029 P006
SFTON3D P029
SMOVL C00154 BC00154 V=166.7  +MOVJ EC00154
SFTOF3D
MOVL C00155 BC00155 V=333.3  +MOVJ EC00155 VJ=30.00
MOVL C00156 BC00156 V=333.3  +MOVJ EC00156 VJ=30.00
MOVL C00157 BC00157 V=333.3  +MOVJ EC00157 VJ=30.00
MOVL C00158 BC00158 V=333.3  +MOVJ EC00158 VJ=30.00
MOVL C00159 BC00159 V=333.3  +MOVJ EC00159 VJ=30.00
SMOVL C00160 BC00160 V=166.7  +MOVJ EC00160
SREFP 3 C00161 BC00161  +REFP EC00161
CALL JOB:SEARCH-R1-S13D
SET P022 P006
SFTON3D P022
SMOVL C00162 BC00162 V=166.7  +MOVJ EC00162
SREFP 3 C00163 BC00163  +REFP EC00163
CALL JOB:SEARCH-R1-S13D
SET P022 P006
SFTON3D P022
SMOVL C00164 BC00164 V=166.7  +MOVJ EC00164
SFTOF3D
MOVL C00165 BC00165 V=333.3  +MOVJ EC00165 VJ=30.00
SMOVL C00166 BC00166 V=166.7  +MOVJ EC00166
SREFP 3 C00167 BC00167  +REFP EC00167
CALL JOB:SEARCH-R1-S13D
SET P021 P006
SFTON3D P021
SMOVL C00168 BC00168 V=166.7  +MOVJ EC00168
SREFP 3 C00169 BC00169  +REFP EC00169
CALL JOB:SEARCH-R1-S13D
SET P021 P006
SFTON3D P021
SMOVL C00170 BC00170 V=166.7  +MOVJ EC00170
MACRO1 MJ#(0) ARGF9
SMOVL C00171 BC00171 V=166.7  +MOVJ EC00171
ARCON
SMOVL C00172 BC00172 V=10.0  +MOVJ EC00172
SMOVL C00173 BC00173 V=10.0  +MOVJ EC00173
SFTON3D P022
SMOVL C00174 BC00174 V=10.0  +MOVJ EC00174
SMOVL C00175 BC00175 V=10.0  +MOVJ EC00175
SMOVL C00176 BC00176 V=10.0  +MOVJ EC00176
ARCOF
SFTOF3D
SMOVL C00177 BC00177 V=250.0  +MOVJ EC00177
SMOVL C00178 BC00178 V=250.0  +MOVJ EC00178
MOVJ C00179 BC00179 VJ=30.00  +MOVJ EC00179 VJ=30.00
MOVJ C00180 BC00180 VJ=30.00  +MOVJ EC00180 VJ=30.00
MOVJ C00181 BC00181 VJ=30.00  +MOVJ EC00181 VJ=30.00
SMOVL C00182 BC00182 V=250.0  +MOVJ EC00182
SFTON3D P029
SMOVL C00183 BC00183 V=250.0  +MOVJ EC00183
ARCON
SMOVL C00184 BC00184 V=10.0  +MOVJ EC00184
SMOVL C00185 BC00185 V=10.0  +MOVJ EC00185
SMOVL C00186 BC00186 V=10.0  +MOVJ EC00186
SMOVL C00187 BC00187 V=10.0  +MOVJ EC00187
ARCOF
SFTOF3D
SMOVL C00188 BC00188 V=333.3  +MOVJ EC00188
SFTON3D P028
SMOVL C00189 BC00189 V=250.0  +MOVJ EC00189
ARCON
SMOVL C00190 BC00190 V=10.0  +MOVJ EC00190
SMOVL C00191 BC00191 V=10.0  +MOVJ EC00191
SMOVL C00192 BC00192 V=10.0  +MOVJ EC00192
SFTON3D P023
SMOVL C00193 BC00193 V=10.0  +MOVJ EC00193
SMOVL C00194 BC00194 V=10.0  +MOVJ EC00194
ARCOF
SFTOF3D
SMOVL C00195 BC00195 V=333.3  +MOVJ EC00195
SFTON3D P024
SMOVL C00196 BC00196 V=166.7  +MOVJ EC00196
ARCON
SMOVL C00197 BC00197 V=10.0  +MOVJ EC00197
SMOVL C00198 BC00198 V=10.0  +MOVJ EC00198
SMOVL C00199 BC00199 V=10.0  +MOVJ EC00199
SMOVL C00200 BC00200 V=10.0  +MOVJ EC00200
SMOVL C00201 BC00201 V=10.0  +MOVJ EC00201
ARCOF
SFTOF3D
SMOVL C00202 BC00202 V=250.0  +MOVJ EC00202
SMOVL C00203 BC00203 V=250.0  +MOVJ EC00203
SFTON3D P026
SMOVL C00204 BC00204 V=250.0  +MOVJ EC00204
ARCON
SMOVL C00205 BC00205 V=10.0  +MOVJ EC00205
SMOVL C00206 BC00206 V=10.0  +MOVJ EC00206
SFTON3D P025
SMOVL C00207 BC00207 V=10.0  +MOVJ EC00207
SMOVL C00208 BC00208 V=10.0  +MOVJ EC00208
SMOVL C00209 BC00209 V=10.0  +MOVJ EC00209
ARCOF
SFTOF3D
SMOVL C00210 BC00210 V=250.0  +MOVJ EC00210
SMOVL C00211 BC00211 V=250.0  +MOVJ EC00211
SFTON3D P027
SMOVL C00212 BC00212 V=250.0  +MOVJ EC00212
ARCON
SMOVL C00213 BC00213 V=10.0  +MOVJ EC00213
SMOVL C00214 BC00214 V=10.0  +MOVJ EC00214
SMOVL C00215 BC00215 V=10.0  +MOVJ EC00215
SMOVL C00216 BC00216 V=10.0  +MOVJ EC00216
SMOVL C00217 BC00217 V=10.0  +MOVJ EC00217
SMOVL C00218 BC00218 V=10.0  +MOVJ EC00218
ARCOF
SFTOF3D
SMOVL C00219 BC00219 V=250.0  +MOVJ EC00219
SMOVL C00220 BC00220 V=250.0  +MOVJ EC00220
MOVJ C00221 BC00221 VJ=30.00  +MOVJ EC00221 VJ=30.00
MOVJ C00222 BC00222 VJ=100.00  +MOVJ EC00222 VJ=100.00
MOVJ C00223 BC00223 VJ=100.00  +MOVJ EC00223 VJ=100.00
END
